Universal Robots PolyScope program: Cooperation_Polishing.urp

Program Cooperation_Polishing (installation=Cooperation_Polishing directory=/home/cobot/ursim-5.11.5.1010327/programs createdIn=5.11.5.1010327 lastSavedIn=5.11.5.1010327 robotSerialNumber=20195599999)
Calibrated DH parameters: a=[0, -0.425, -0.3922, 0, 0, 0]; d=[0.1625, 0, 0, 0.1333, 0.0997, 0.0996]; alpha=[1.570796, 0, 0, 1.570796, -1.570796, 0]; deltaTheta=[0, 0, 0, 0, 0, 0]
Robot Program (runOnlyOnce=false)
  Wait DigitalInput pin=ib64; digitalValue=1
  Switch expression=GP_int_in[24]
    Case (caseValue=1)
      'Move to Home position'
      SafeHome (positionOptionType=SPEED_AND_ACCELERATION speed=1.047198 acceleration=1.396263 nextMotionTime=2)
    Case (caseValue=2)
      'Read startPos, endPos'
      startPos := p[if24_x,if25_y,if26_z,if27_rx,if28_ry,if29_rz]
      endPos := p[GP_float_in[30],GP_float_in[31],GP_float_in[32],GP_float_in[33],GP_float_in[34],GP_float_in[35]]
      'Move: startPos -> endPos -> startPos'
      MoveL speed 100 mm/s, acceleration 500 mm/s^2 (useActiveTCP=true) feature=Surface
        Waypoint Waypoint (Variable): variable=startPos
        Waypoint Waypoint (Variable): variable=endPos
        Waypoint Waypoint (Variable): variable=startPos
    Case (caseValue=2147483647)
      'Do nothing (just handshake)'
  Set DigitalOutput pin=ob64; digitalValue=1
  Wait DigitalInput pin=ib64; digitalValue=0
  Set DigitalOutput pin=ob64; digitalValue=0
